FUNCTION_BLOCK F_CONCAT_DATE_TOD (* concatenation *)
  (* Standard: 61131-3; Classification: standard function of character string *)
  (* Version 0.0, 2013-04-25, 4DIAC-IDE, 4DIAC-Consortium *)
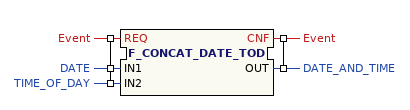
  EVENT_INPUT
    REQ WITH IN1, IN2; (* Service Request *)
  END_EVENT
  EVENT_OUTPUT
    CNF WITH OUT; (* Confirmation of Requested Service *)
  END_EVENT
  VAR_INPUT
    IN1 : DATE; (* input string 1 *)
    IN2 : TIME_OF_DAY; (* input string 2 *)
  END_VAR
  VAR_OUTPUT
    OUT : DATE_AND_TIME; (* date + time of day *)
  END_VAR
END_FUNCTION_BLOCK
